// TIA Portal V17 export
// export: Created 2023-03-24T09:45:04.5136241Z, ExportSetting None, DisplayName Totally Integrated Automation Portal, DisplayVersion V17 Update 4, DisplayName TIA Portal Openness, DisplayVersion V17 Update 4, DisplayName TIA Portal Version Control Interface, DisplayVersion V17, DisplayName STEP 7 Professional, DisplayVersion V17 Update 4, DisplayName STEP 7 Safety, DisplayVersion V17, DisplayName WinCC Advanced / Unified PC, DisplayVersion V17 Update 4
FUNCTION "FC_PROVA" : Void   // FC1, LAD
TITLE = goku
{ S7_Optimized_Access := 'TRUE' }
// bigol
// stored: SetENOAutomatically false
BEGIN

REGION Network 1: BYPASS CONTROL VALVE OVER 1ST-3RD STAGE OPEN
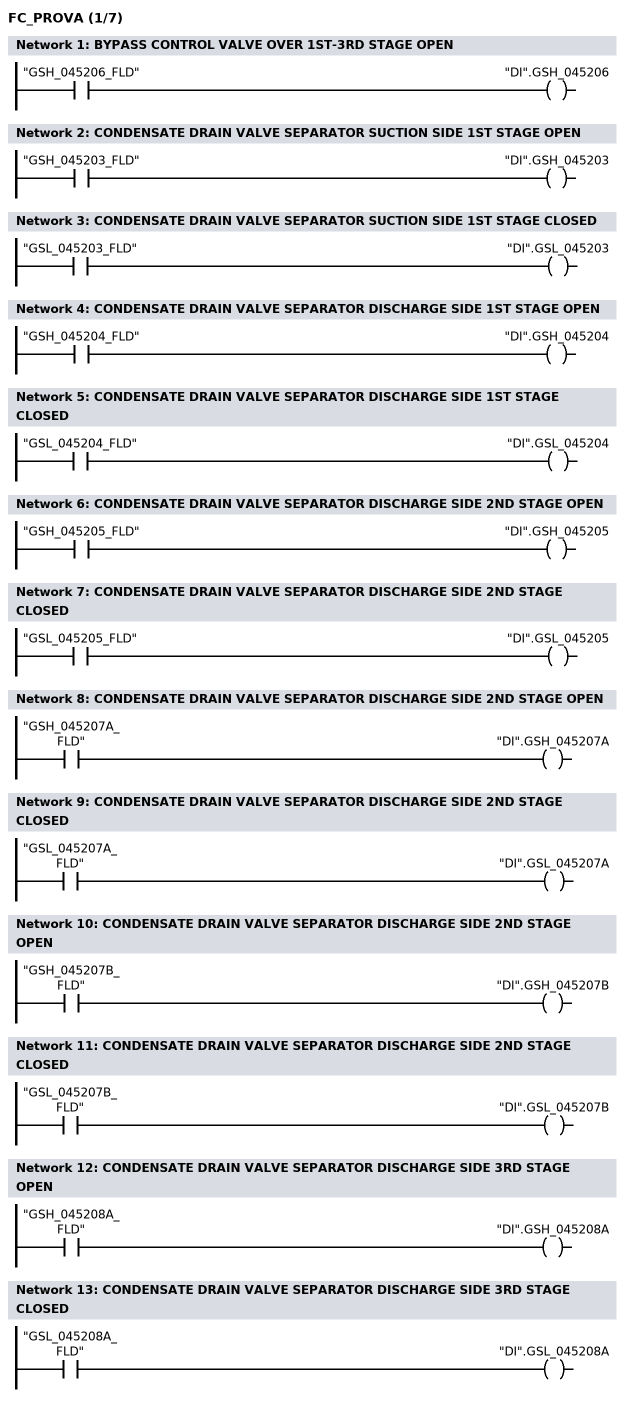
   RUNG wire#powerrail
      Contact( "GSH_045206_FLD" )
      Coil( "DI".GSH_045206 )
   END_RUNG
   // the same network as SCL:
   "DI".GSH_045206 := "GSH_045206_FLD";
END_REGION

REGION Network 2: CONDENSATE DRAIN VALVE SEPARATOR SUCTION SIDE 1ST STAGE OPEN
   RUNG wire#powerrail
      Contact( "GSH_045203_FLD" )
      Coil( "DI".GSH_045203 )
   END_RUNG
   // the same network as SCL:
   "DI".GSH_045203 := "GSH_045203_FLD";
END_REGION

REGION Network 3: CONDENSATE DRAIN VALVE SEPARATOR SUCTION SIDE 1ST STAGE CLOSED
   RUNG wire#powerrail
      Contact( "GSL_045203_FLD" )
      Coil( "DI".GSL_045203 )
   END_RUNG
   // the same network as SCL:
   "DI".GSL_045203 := "GSL_045203_FLD";
END_REGION

REGION Network 4: CONDENSATE DRAIN VALVE SEPARATOR DISCHARGE SIDE 1ST STAGE OPEN
   RUNG wire#powerrail
      Contact( "GSH_045204_FLD" )
      Coil( "DI".GSH_045204 )
   END_RUNG
   // the same network as SCL:
   "DI".GSH_045204 := "GSH_045204_FLD";
END_REGION

REGION Network 5: CONDENSATE DRAIN VALVE SEPARATOR DISCHARGE SIDE 1ST STAGE CLOSED
   RUNG wire#powerrail
      Contact( "GSL_045204_FLD" )
      Coil( "DI".GSL_045204 )
   END_RUNG
   // the same network as SCL:
   "DI".GSL_045204 := "GSL_045204_FLD";
END_REGION

REGION Network 6: CONDENSATE DRAIN VALVE SEPARATOR DISCHARGE SIDE 2ND STAGE OPEN
   RUNG wire#powerrail
      Contact( "GSH_045205_FLD" )
      Coil( "DI".GSH_045205 )
   END_RUNG
   // the same network as SCL:
   "DI".GSH_045205 := "GSH_045205_FLD";
END_REGION

REGION Network 7: CONDENSATE DRAIN VALVE SEPARATOR DISCHARGE SIDE 2ND STAGE CLOSED
   RUNG wire#powerrail
      Contact( "GSL_045205_FLD" )
      Coil( "DI".GSL_045205 )
   END_RUNG
   // the same network as SCL:
   "DI".GSL_045205 := "GSL_045205_FLD";
END_REGION

REGION Network 8: CONDENSATE DRAIN VALVE SEPARATOR DISCHARGE SIDE 2ND STAGE OPEN
   RUNG wire#powerrail
      Contact( "GSH_045207A_FLD" )
      Coil( "DI".GSH_045207A )
   END_RUNG
   // the same network as SCL:
   "DI".GSH_045207A := "GSH_045207A_FLD";
END_REGION

REGION Network 9: CONDENSATE DRAIN VALVE SEPARATOR DISCHARGE SIDE 2ND STAGE CLOSED
   RUNG wire#powerrail
      Contact( "GSL_045207A_FLD" )
      Coil( "DI".GSL_045207A )
   END_RUNG
   // the same network as SCL:
   "DI".GSL_045207A := "GSL_045207A_FLD";
END_REGION

REGION Network 10: CONDENSATE DRAIN VALVE SEPARATOR DISCHARGE SIDE 2ND STAGE OPEN
   RUNG wire#powerrail
      Contact( "GSH_045207B_FLD" )
      Coil( "DI".GSH_045207B )
   END_RUNG
   // the same network as SCL:
   "DI".GSH_045207B := "GSH_045207B_FLD";
END_REGION

REGION Network 11: CONDENSATE DRAIN VALVE SEPARATOR DISCHARGE SIDE 2ND STAGE CLOSED
   RUNG wire#powerrail
      Contact( "GSL_045207B_FLD" )
      Coil( "DI".GSL_045207B )
   END_RUNG
   // the same network as SCL:
   "DI".GSL_045207B := "GSL_045207B_FLD";
END_REGION

REGION Network 12: CONDENSATE DRAIN VALVE SEPARATOR DISCHARGE SIDE 3RD STAGE OPEN
   RUNG wire#powerrail
      Contact( "GSH_045208A_FLD" )
      Coil( "DI".GSH_045208A )
   END_RUNG
   // the same network as SCL:
   "DI".GSH_045208A := "GSH_045208A_FLD";
END_REGION

REGION Network 13: CONDENSATE DRAIN VALVE SEPARATOR DISCHARGE SIDE 3RD STAGE CLOSED
   RUNG wire#powerrail
      Contact( "GSL_045208A_FLD" )
      Coil( "DI".GSL_045208A )
   END_RUNG
   // the same network as SCL:
   "DI".GSL_045208A := "GSL_045208A_FLD";
END_REGION

REGION Network 14: CONDENSATE DRAIN VALVE SEPARATOR DISCHARGE SIDE 3RD STAGE OPEN
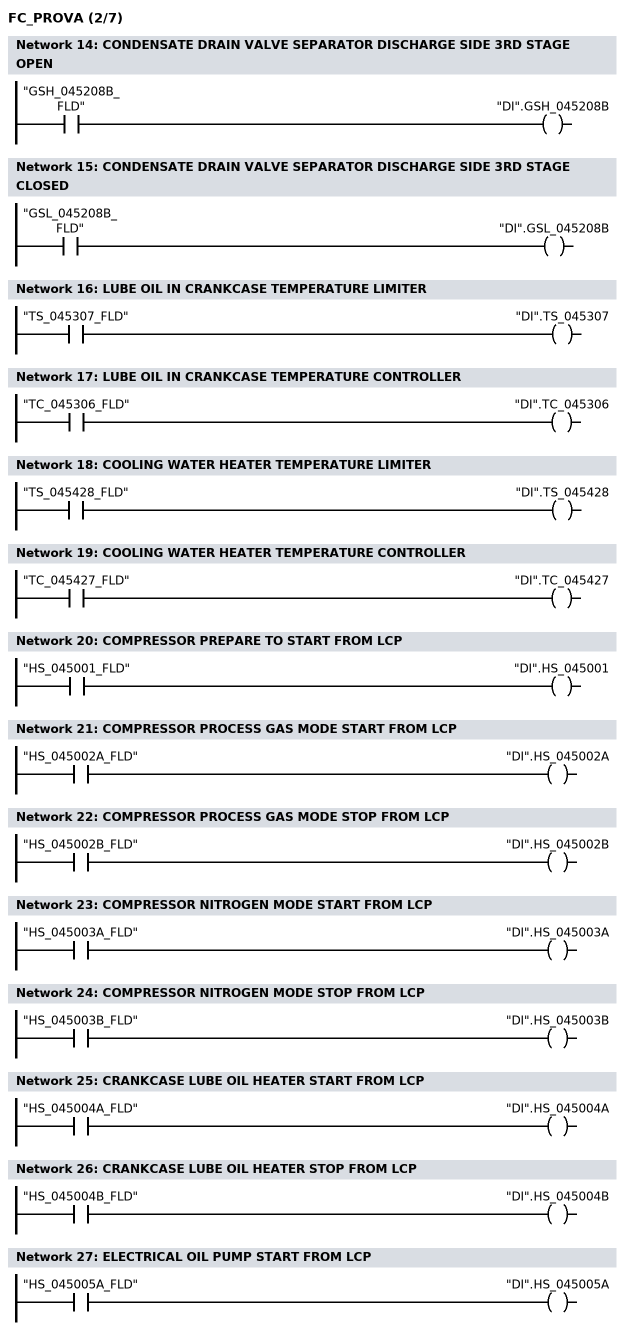
   RUNG wire#powerrail
      Contact( "GSH_045208B_FLD" )
      Coil( "DI".GSH_045208B )
   END_RUNG
   // the same network as SCL:
   "DI".GSH_045208B := "GSH_045208B_FLD";
END_REGION

REGION Network 15: CONDENSATE DRAIN VALVE SEPARATOR DISCHARGE SIDE 3RD STAGE CLOSED
   RUNG wire#powerrail
      Contact( "GSL_045208B_FLD" )
      Coil( "DI".GSL_045208B )
   END_RUNG
   // the same network as SCL:
   "DI".GSL_045208B := "GSL_045208B_FLD";
END_REGION

REGION Network 16: LUBE OIL IN CRANKCASE TEMPERATURE LIMITER
   RUNG wire#powerrail
      Contact( "TS_045307_FLD" )
      Coil( "DI".TS_045307 )
   END_RUNG
   // the same network as SCL:
   "DI".TS_045307 := "TS_045307_FLD";
END_REGION

REGION Network 17: LUBE OIL IN CRANKCASE TEMPERATURE CONTROLLER
   RUNG wire#powerrail
      Contact( "TC_045306_FLD" )
      Coil( "DI".TC_045306 )
   END_RUNG
   // the same network as SCL:
   "DI".TC_045306 := "TC_045306_FLD";
END_REGION

REGION Network 18: COOLING WATER HEATER TEMPERATURE LIMITER
   RUNG wire#powerrail
      Contact( "TS_045428_FLD" )
      Coil( "DI".TS_045428 )
   END_RUNG
   // the same network as SCL:
   "DI".TS_045428 := "TS_045428_FLD";
END_REGION

REGION Network 19: COOLING WATER HEATER TEMPERATURE CONTROLLER
   RUNG wire#powerrail
      Contact( "TC_045427_FLD" )
      Coil( "DI".TC_045427 )
   END_RUNG
   // the same network as SCL:
   "DI".TC_045427 := "TC_045427_FLD";
END_REGION

REGION Network 20: COMPRESSOR PREPARE TO START FROM LCP
   RUNG wire#powerrail
      Contact( "HS_045001_FLD" )
      Coil( "DI".HS_045001 )
   END_RUNG
   // the same network as SCL:
   "DI".HS_045001 := "HS_045001_FLD";
END_REGION

REGION Network 21: COMPRESSOR PROCESS GAS MODE START FROM LCP
   RUNG wire#powerrail
      Contact( "HS_045002A_FLD" )
      Coil( "DI".HS_045002A )
   END_RUNG
   // the same network as SCL:
   "DI".HS_045002A := "HS_045002A_FLD";
END_REGION

REGION Network 22: COMPRESSOR PROCESS GAS MODE STOP FROM LCP
   RUNG wire#powerrail
      Contact( "HS_045002B_FLD" )
      Coil( "DI".HS_045002B )
   END_RUNG
   // the same network as SCL:
   "DI".HS_045002B := "HS_045002B_FLD";
END_REGION

REGION Network 23: COMPRESSOR NITROGEN MODE START FROM LCP
   RUNG wire#powerrail
      Contact( "HS_045003A_FLD" )
      Coil( "DI".HS_045003A )
   END_RUNG
   // the same network as SCL:
   "DI".HS_045003A := "HS_045003A_FLD";
END_REGION

REGION Network 24: COMPRESSOR NITROGEN MODE STOP FROM LCP
   RUNG wire#powerrail
      Contact( "HS_045003B_FLD" )
      Coil( "DI".HS_045003B )
   END_RUNG
   // the same network as SCL:
   "DI".HS_045003B := "HS_045003B_FLD";
END_REGION

REGION Network 25: CRANKCASE LUBE OIL HEATER START FROM LCP
   RUNG wire#powerrail
      Contact( "HS_045004A_FLD" )
      Coil( "DI".HS_045004A )
   END_RUNG
   // the same network as SCL:
   "DI".HS_045004A := "HS_045004A_FLD";
END_REGION

REGION Network 26: CRANKCASE LUBE OIL HEATER STOP FROM LCP
   RUNG wire#powerrail
      Contact( "HS_045004B_FLD" )
      Coil( "DI".HS_045004B )
   END_RUNG
   // the same network as SCL:
   "DI".HS_045004B := "HS_045004B_FLD";
END_REGION

REGION Network 27: ELECTRICAL OIL PUMP START FROM LCP
   RUNG wire#powerrail
      Contact( "HS_045005A_FLD" )
      Coil( "DI".HS_045005A )
   END_RUNG
   // the same network as SCL:
   "DI".HS_045005A := "HS_045005A_FLD";
END_REGION

REGION Network 28: ELECTRICAL OIL PUMP STOP FROM LCP
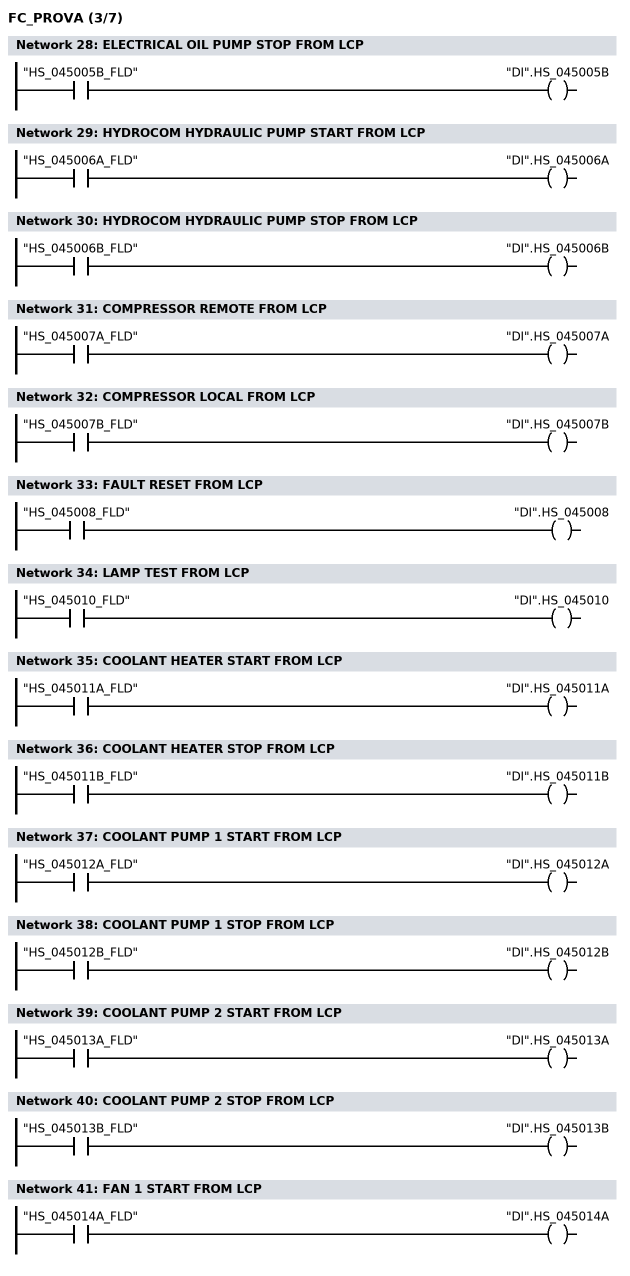
   RUNG wire#powerrail
      Contact( "HS_045005B_FLD" )
      Coil( "DI".HS_045005B )
   END_RUNG
   // the same network as SCL:
   "DI".HS_045005B := "HS_045005B_FLD";
END_REGION

REGION Network 29: HYDROCOM HYDRAULIC PUMP START FROM LCP
   RUNG wire#powerrail
      Contact( "HS_045006A_FLD" )
      Coil( "DI".HS_045006A )
   END_RUNG
   // the same network as SCL:
   "DI".HS_045006A := "HS_045006A_FLD";
END_REGION

REGION Network 30: HYDROCOM HYDRAULIC PUMP STOP FROM LCP
   RUNG wire#powerrail
      Contact( "HS_045006B_FLD" )
      Coil( "DI".HS_045006B )
   END_RUNG
   // the same network as SCL:
   "DI".HS_045006B := "HS_045006B_FLD";
END_REGION

REGION Network 31: COMPRESSOR REMOTE FROM LCP
   RUNG wire#powerrail
      Contact( "HS_045007A_FLD" )
      Coil( "DI".HS_045007A )
   END_RUNG
   // the same network as SCL:
   "DI".HS_045007A := "HS_045007A_FLD";
END_REGION

REGION Network 32: COMPRESSOR LOCAL FROM LCP
   RUNG wire#powerrail
      Contact( "HS_045007B_FLD" )
      Coil( "DI".HS_045007B )
   END_RUNG
   // the same network as SCL:
   "DI".HS_045007B := "HS_045007B_FLD";
END_REGION

REGION Network 33: FAULT RESET FROM LCP
   RUNG wire#powerrail
      Contact( "HS_045008_FLD" )
      Coil( "DI".HS_045008 )
   END_RUNG
   // the same network as SCL:
   "DI".HS_045008 := "HS_045008_FLD";
END_REGION

REGION Network 34: LAMP TEST FROM LCP
   RUNG wire#powerrail
      Contact( "HS_045010_FLD" )
      Coil( "DI".HS_045010 )
   END_RUNG
   // the same network as SCL:
   "DI".HS_045010 := "HS_045010_FLD";
END_REGION

REGION Network 35: COOLANT HEATER START FROM LCP
   RUNG wire#powerrail
      Contact( "HS_045011A_FLD" )
      Coil( "DI".HS_045011A )
   END_RUNG
   // the same network as SCL:
   "DI".HS_045011A := "HS_045011A_FLD";
END_REGION

REGION Network 36: COOLANT HEATER STOP FROM LCP
   RUNG wire#powerrail
      Contact( "HS_045011B_FLD" )
      Coil( "DI".HS_045011B )
   END_RUNG
   // the same network as SCL:
   "DI".HS_045011B := "HS_045011B_FLD";
END_REGION

REGION Network 37: COOLANT PUMP 1 START FROM LCP
   RUNG wire#powerrail
      Contact( "HS_045012A_FLD" )
      Coil( "DI".HS_045012A )
   END_RUNG
   // the same network as SCL:
   "DI".HS_045012A := "HS_045012A_FLD";
END_REGION

REGION Network 38: COOLANT PUMP 1 STOP FROM LCP
   RUNG wire#powerrail
      Contact( "HS_045012B_FLD" )
      Coil( "DI".HS_045012B )
   END_RUNG
   // the same network as SCL:
   "DI".HS_045012B := "HS_045012B_FLD";
END_REGION

REGION Network 39: COOLANT PUMP 2 START FROM LCP
   RUNG wire#powerrail
      Contact( "HS_045013A_FLD" )
      Coil( "DI".HS_045013A )
   END_RUNG
   // the same network as SCL:
   "DI".HS_045013A := "HS_045013A_FLD";
END_REGION

REGION Network 40: COOLANT PUMP 2 STOP FROM LCP
   RUNG wire#powerrail
      Contact( "HS_045013B_FLD" )
      Coil( "DI".HS_045013B )
   END_RUNG
   // the same network as SCL:
   "DI".HS_045013B := "HS_045013B_FLD";
END_REGION

REGION Network 41: FAN 1 START FROM LCP
   RUNG wire#powerrail
      Contact( "HS_045014A_FLD" )
      Coil( "DI".HS_045014A )
   END_RUNG
   // the same network as SCL:
   "DI".HS_045014A := "HS_045014A_FLD";
END_REGION

REGION Network 42: FAN 1 STOP FROM LCP
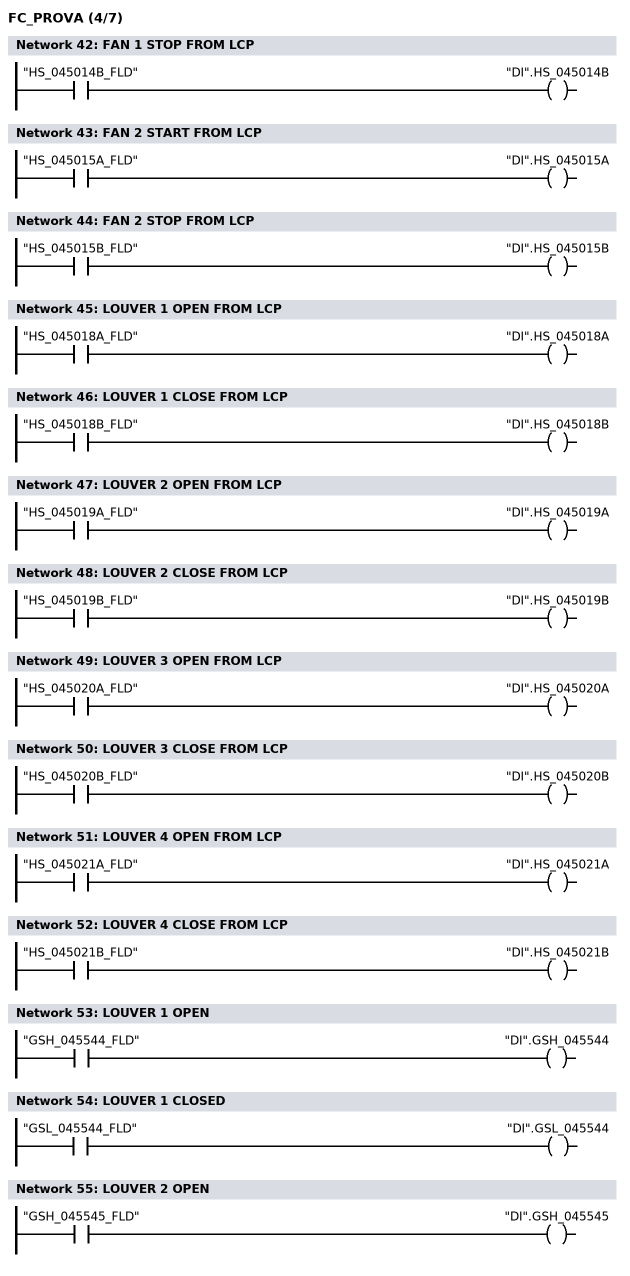
   RUNG wire#powerrail
      Contact( "HS_045014B_FLD" )
      Coil( "DI".HS_045014B )
   END_RUNG
   // the same network as SCL:
   "DI".HS_045014B := "HS_045014B_FLD";
END_REGION

REGION Network 43: FAN 2 START FROM LCP
   RUNG wire#powerrail
      Contact( "HS_045015A_FLD" )
      Coil( "DI".HS_045015A )
   END_RUNG
   // the same network as SCL:
   "DI".HS_045015A := "HS_045015A_FLD";
END_REGION

REGION Network 44: FAN 2 STOP FROM LCP
   RUNG wire#powerrail
      Contact( "HS_045015B_FLD" )
      Coil( "DI".HS_045015B )
   END_RUNG
   // the same network as SCL:
   "DI".HS_045015B := "HS_045015B_FLD";
END_REGION

REGION Network 45: LOUVER 1 OPEN FROM LCP
   RUNG wire#powerrail
      Contact( "HS_045018A_FLD" )
      Coil( "DI".HS_045018A )
   END_RUNG
   // the same network as SCL:
   "DI".HS_045018A := "HS_045018A_FLD";
END_REGION

REGION Network 46: LOUVER 1 CLOSE FROM LCP
   RUNG wire#powerrail
      Contact( "HS_045018B_FLD" )
      Coil( "DI".HS_045018B )
   END_RUNG
   // the same network as SCL:
   "DI".HS_045018B := "HS_045018B_FLD";
END_REGION

REGION Network 47: LOUVER 2 OPEN FROM LCP
   RUNG wire#powerrail
      Contact( "HS_045019A_FLD" )
      Coil( "DI".HS_045019A )
   END_RUNG
   // the same network as SCL:
   "DI".HS_045019A := "HS_045019A_FLD";
END_REGION

REGION Network 48: LOUVER 2 CLOSE FROM LCP
   RUNG wire#powerrail
      Contact( "HS_045019B_FLD" )
      Coil( "DI".HS_045019B )
   END_RUNG
   // the same network as SCL:
   "DI".HS_045019B := "HS_045019B_FLD";
END_REGION

REGION Network 49: LOUVER 3 OPEN FROM LCP
   RUNG wire#powerrail
      Contact( "HS_045020A_FLD" )
      Coil( "DI".HS_045020A )
   END_RUNG
   // the same network as SCL:
   "DI".HS_045020A := "HS_045020A_FLD";
END_REGION

REGION Network 50: LOUVER 3 CLOSE FROM LCP
   RUNG wire#powerrail
      Contact( "HS_045020B_FLD" )
      Coil( "DI".HS_045020B )
   END_RUNG
   // the same network as SCL:
   "DI".HS_045020B := "HS_045020B_FLD";
END_REGION

REGION Network 51: LOUVER 4 OPEN FROM LCP
   RUNG wire#powerrail
      Contact( "HS_045021A_FLD" )
      Coil( "DI".HS_045021A )
   END_RUNG
   // the same network as SCL:
   "DI".HS_045021A := "HS_045021A_FLD";
END_REGION

REGION Network 52: LOUVER 4 CLOSE FROM LCP
   RUNG wire#powerrail
      Contact( "HS_045021B_FLD" )
      Coil( "DI".HS_045021B )
   END_RUNG
   // the same network as SCL:
   "DI".HS_045021B := "HS_045021B_FLD";
END_REGION

REGION Network 53: LOUVER 1 OPEN
   RUNG wire#powerrail
      Contact( "GSH_045544_FLD" )
      Coil( "DI".GSH_045544 )
   END_RUNG
   // the same network as SCL:
   "DI".GSH_045544 := "GSH_045544_FLD";
END_REGION

REGION Network 54: LOUVER 1 CLOSED
   RUNG wire#powerrail
      Contact( "GSL_045544_FLD" )
      Coil( "DI".GSL_045544 )
   END_RUNG
   // the same network as SCL:
   "DI".GSL_045544 := "GSL_045544_FLD";
END_REGION

REGION Network 55: LOUVER 2 OPEN
   RUNG wire#powerrail
      Contact( "GSH_045545_FLD" )
      Coil( "DI".GSH_045545 )
   END_RUNG
   // the same network as SCL:
   "DI".GSH_045545 := "GSH_045545_FLD";
END_REGION

REGION Network 56: LOUVER 2 CLOSED
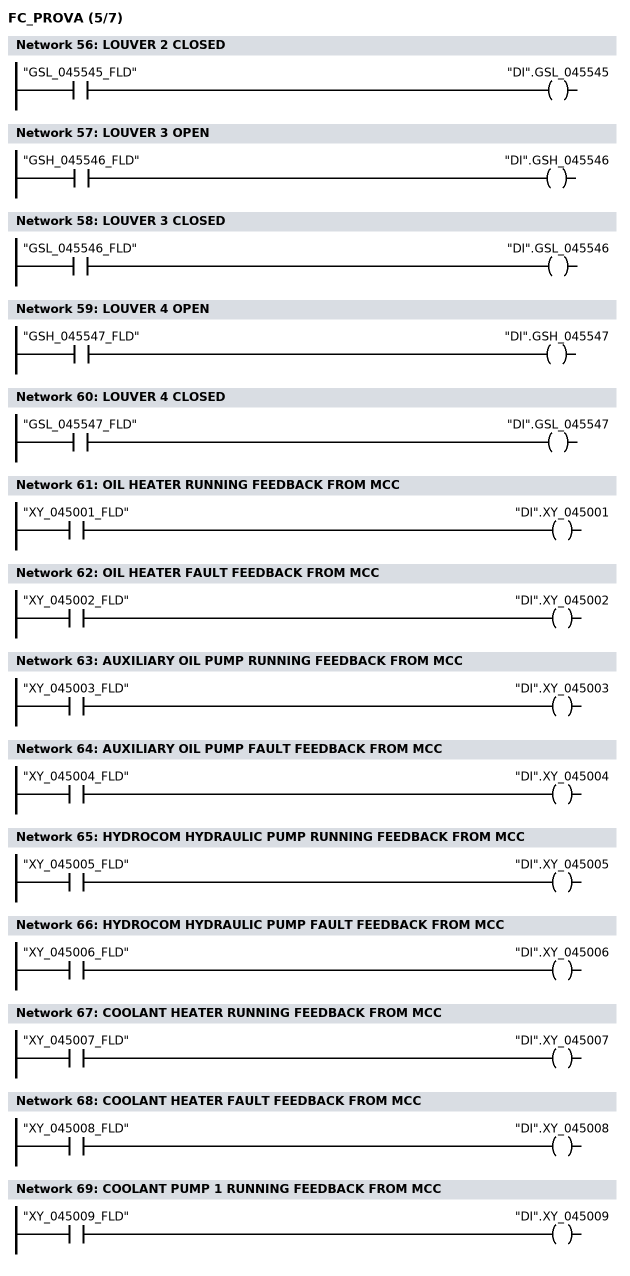
   RUNG wire#powerrail
      Contact( "GSL_045545_FLD" )
      Coil( "DI".GSL_045545 )
   END_RUNG
   // the same network as SCL:
   "DI".GSL_045545 := "GSL_045545_FLD";
END_REGION

REGION Network 57: LOUVER 3 OPEN
   RUNG wire#powerrail
      Contact( "GSH_045546_FLD" )
      Coil( "DI".GSH_045546 )
   END_RUNG
   // the same network as SCL:
   "DI".GSH_045546 := "GSH_045546_FLD";
END_REGION

REGION Network 58: LOUVER 3 CLOSED
   RUNG wire#powerrail
      Contact( "GSL_045546_FLD" )
      Coil( "DI".GSL_045546 )
   END_RUNG
   // the same network as SCL:
   "DI".GSL_045546 := "GSL_045546_FLD";
END_REGION

REGION Network 59: LOUVER 4 OPEN
   RUNG wire#powerrail
      Contact( "GSH_045547_FLD" )
      Coil( "DI".GSH_045547 )
   END_RUNG
   // the same network as SCL:
   "DI".GSH_045547 := "GSH_045547_FLD";
END_REGION

REGION Network 60: LOUVER 4 CLOSED
   RUNG wire#powerrail
      Contact( "GSL_045547_FLD" )
      Coil( "DI".GSL_045547 )
   END_RUNG
   // the same network as SCL:
   "DI".GSL_045547 := "GSL_045547_FLD";
END_REGION

REGION Network 61: OIL HEATER RUNNING FEEDBACK FROM MCC
   RUNG wire#powerrail
      Contact( "XY_045001_FLD" )
      Coil( "DI".XY_045001 )
   END_RUNG
   // the same network as SCL:
   "DI".XY_045001 := "XY_045001_FLD";
END_REGION

REGION Network 62: OIL HEATER FAULT FEEDBACK FROM MCC
   RUNG wire#powerrail
      Contact( "XY_045002_FLD" )
      Coil( "DI".XY_045002 )
   END_RUNG
   // the same network as SCL:
   "DI".XY_045002 := "XY_045002_FLD";
END_REGION

REGION Network 63: AUXILIARY OIL PUMP RUNNING FEEDBACK FROM MCC
   RUNG wire#powerrail
      Contact( "XY_045003_FLD" )
      Coil( "DI".XY_045003 )
   END_RUNG
   // the same network as SCL:
   "DI".XY_045003 := "XY_045003_FLD";
END_REGION

REGION Network 64: AUXILIARY OIL PUMP FAULT FEEDBACK FROM MCC
   RUNG wire#powerrail
      Contact( "XY_045004_FLD" )
      Coil( "DI".XY_045004 )
   END_RUNG
   // the same network as SCL:
   "DI".XY_045004 := "XY_045004_FLD";
END_REGION

REGION Network 65: HYDROCOM HYDRAULIC PUMP RUNNING FEEDBACK FROM MCC
   RUNG wire#powerrail
      Contact( "XY_045005_FLD" )
      Coil( "DI".XY_045005 )
   END_RUNG
   // the same network as SCL:
   "DI".XY_045005 := "XY_045005_FLD";
END_REGION

REGION Network 66: HYDROCOM HYDRAULIC PUMP FAULT FEEDBACK FROM MCC
   RUNG wire#powerrail
      Contact( "XY_045006_FLD" )
      Coil( "DI".XY_045006 )
   END_RUNG
   // the same network as SCL:
   "DI".XY_045006 := "XY_045006_FLD";
END_REGION

REGION Network 67: COOLANT HEATER RUNNING FEEDBACK FROM MCC
   RUNG wire#powerrail
      Contact( "XY_045007_FLD" )
      Coil( "DI".XY_045007 )
   END_RUNG
   // the same network as SCL:
   "DI".XY_045007 := "XY_045007_FLD";
END_REGION

REGION Network 68: COOLANT HEATER FAULT FEEDBACK FROM MCC
   RUNG wire#powerrail
      Contact( "XY_045008_FLD" )
      Coil( "DI".XY_045008 )
   END_RUNG
   // the same network as SCL:
   "DI".XY_045008 := "XY_045008_FLD";
END_REGION

REGION Network 69: COOLANT PUMP 1 RUNNING FEEDBACK FROM MCC
   RUNG wire#powerrail
      Contact( "XY_045009_FLD" )
      Coil( "DI".XY_045009 )
   END_RUNG
   // the same network as SCL:
   "DI".XY_045009 := "XY_045009_FLD";
END_REGION

REGION Network 70: COOLANT PUMP 1 FAULT FEEDBACK FROM MCC
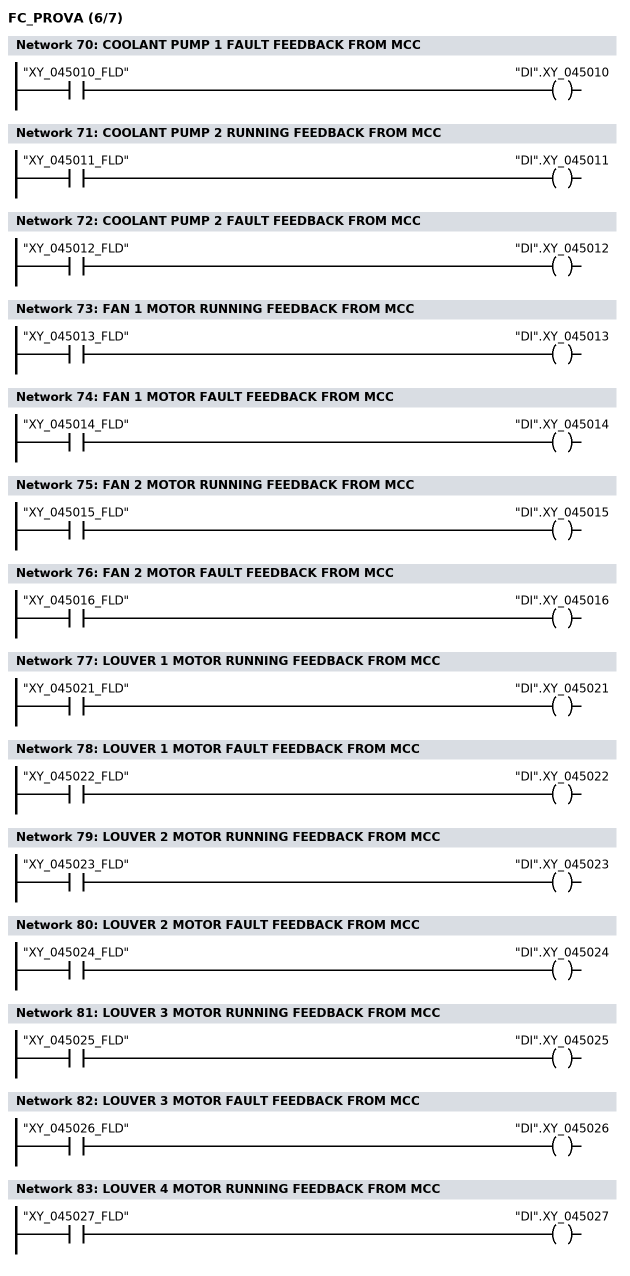
   RUNG wire#powerrail
      Contact( "XY_045010_FLD" )
      Coil( "DI".XY_045010 )
   END_RUNG
   // the same network as SCL:
   "DI".XY_045010 := "XY_045010_FLD";
END_REGION

REGION Network 71: COOLANT PUMP 2 RUNNING FEEDBACK FROM MCC
   RUNG wire#powerrail
      Contact( "XY_045011_FLD" )
      Coil( "DI".XY_045011 )
   END_RUNG
   // the same network as SCL:
   "DI".XY_045011 := "XY_045011_FLD";
END_REGION

REGION Network 72: COOLANT PUMP 2 FAULT FEEDBACK FROM MCC
   RUNG wire#powerrail
      Contact( "XY_045012_FLD" )
      Coil( "DI".XY_045012 )
   END_RUNG
   // the same network as SCL:
   "DI".XY_045012 := "XY_045012_FLD";
END_REGION

REGION Network 73: FAN 1 MOTOR RUNNING FEEDBACK FROM MCC
   RUNG wire#powerrail
      Contact( "XY_045013_FLD" )
      Coil( "DI".XY_045013 )
   END_RUNG
   // the same network as SCL:
   "DI".XY_045013 := "XY_045013_FLD";
END_REGION

REGION Network 74: FAN 1 MOTOR FAULT FEEDBACK FROM MCC
   RUNG wire#powerrail
      Contact( "XY_045014_FLD" )
      Coil( "DI".XY_045014 )
   END_RUNG
   // the same network as SCL:
   "DI".XY_045014 := "XY_045014_FLD";
END_REGION

REGION Network 75: FAN 2 MOTOR RUNNING FEEDBACK FROM MCC
   RUNG wire#powerrail
      Contact( "XY_045015_FLD" )
      Coil( "DI".XY_045015 )
   END_RUNG
   // the same network as SCL:
   "DI".XY_045015 := "XY_045015_FLD";
END_REGION

REGION Network 76: FAN 2 MOTOR FAULT FEEDBACK FROM MCC
   RUNG wire#powerrail
      Contact( "XY_045016_FLD" )
      Coil( "DI".XY_045016 )
   END_RUNG
   // the same network as SCL:
   "DI".XY_045016 := "XY_045016_FLD";
END_REGION

REGION Network 77: LOUVER 1 MOTOR RUNNING FEEDBACK FROM MCC
   RUNG wire#powerrail
      Contact( "XY_045021_FLD" )
      Coil( "DI".XY_045021 )
   END_RUNG
   // the same network as SCL:
   "DI".XY_045021 := "XY_045021_FLD";
END_REGION

REGION Network 78: LOUVER 1 MOTOR FAULT FEEDBACK FROM MCC
   RUNG wire#powerrail
      Contact( "XY_045022_FLD" )
      Coil( "DI".XY_045022 )
   END_RUNG
   // the same network as SCL:
   "DI".XY_045022 := "XY_045022_FLD";
END_REGION

REGION Network 79: LOUVER 2 MOTOR RUNNING FEEDBACK FROM MCC
   RUNG wire#powerrail
      Contact( "XY_045023_FLD" )
      Coil( "DI".XY_045023 )
   END_RUNG
   // the same network as SCL:
   "DI".XY_045023 := "XY_045023_FLD";
END_REGION

REGION Network 80: LOUVER 2 MOTOR FAULT FEEDBACK FROM MCC
   RUNG wire#powerrail
      Contact( "XY_045024_FLD" )
      Coil( "DI".XY_045024 )
   END_RUNG
   // the same network as SCL:
   "DI".XY_045024 := "XY_045024_FLD";
END_REGION

REGION Network 81: LOUVER 3 MOTOR RUNNING FEEDBACK FROM MCC
   RUNG wire#powerrail
      Contact( "XY_045025_FLD" )
      Coil( "DI".XY_045025 )
   END_RUNG
   // the same network as SCL:
   "DI".XY_045025 := "XY_045025_FLD";
END_REGION

REGION Network 82: LOUVER 3 MOTOR FAULT FEEDBACK FROM MCC
   RUNG wire#powerrail
      Contact( "XY_045026_FLD" )
      Coil( "DI".XY_045026 )
   END_RUNG
   // the same network as SCL:
   "DI".XY_045026 := "XY_045026_FLD";
END_REGION

REGION Network 83: LOUVER 4 MOTOR RUNNING FEEDBACK FROM MCC
   RUNG wire#powerrail
      Contact( "XY_045027_FLD" )
      Coil( "DI".XY_045027 )
   END_RUNG
   // the same network as SCL:
   "DI".XY_045027 := "XY_045027_FLD";
END_REGION

REGION Network 84: LOUVER 4 MOTOR FAULT FEEDBACK FROM MCC
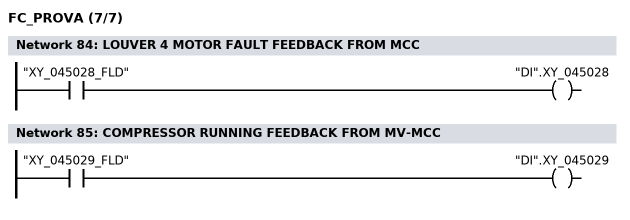
   RUNG wire#powerrail
      Contact( "XY_045028_FLD" )
      Coil( "DI".XY_045028 )
   END_RUNG
   // the same network as SCL:
   "DI".XY_045028 := "XY_045028_FLD";
END_REGION

REGION Network 85: COMPRESSOR RUNNING FEEDBACK FROM MV-MCC
   RUNG wire#powerrail
      Contact( "XY_045029_FLD" )
      Coil( "DI".XY_045029 )
   END_RUNG
   // the same network as SCL:
   "DI".XY_045029 := "XY_045029_FLD";
END_REGION
END_FUNCTION
